FUNCTION_BLOCK FB_Test_Base_Ptr EXTENDS FB_UnitTestBase
VAR_INPUT
END_VAR
VAR_OUTPUT
END_VAR
VAR
END_VAR

(******************************************************************************
Baustein: FB_Test_Base.cleanup
Spezifikation: doc/Spezifikation.pdf, Kap. x.y.z
-------------------------------------------------------------------------------
erstellt:
von:
Geändert:
von:
-------------------------------------------------------------------------------
Beschreibung
Diese Methode...

-------------------------------------------------------------------------------
Input
-

Output
-
******************************************************************************)
METHOD PUBLIC cleanup : BOOL
VAR_INPUT
END_VAR

	cleanup := true;
END_METHOD

(******************************************************************************
Baustein: FB_Test_Base.execute
Spezifikation: doc/Spezifikation.pdf, Kap. x.y.z
-------------------------------------------------------------------------------
erstellt:
von:
Geändert:
von:
-------------------------------------------------------------------------------
Beschreibung
Diese Methode...

-------------------------------------------------------------------------------
Input
-

Output
-
******************************************************************************)
METHOD PUBLIC execute : BOOL
VAR_INPUT
END_VAR
VAR
	bValue1   : ARRAY[0..10] OF BOOL;
	bValue2   : ARRAY[0..10] OF BOOL;
	s8Value1  : ARRAY[0..10] OF SINT;
	s8Value2  : ARRAY[0..10] OF SINT;
	u8Value1  : ARRAY[0..10] OF USINT;
	u8Value2  : ARRAY[0..10] OF USINT;	
	s16Value1 : ARRAY[0..10] OF INT;
	s16Value2 : ARRAY[0..10] OF INT;
	u16Value1 : ARRAY[0..10] OF UINT;
	u16Value2 : ARRAY[0..10] OF UINT;		
	s32Value1 : ARRAY[0..10] OF DINT;
	s32Value2 : ARRAY[0..10] OF DINT;
	u32Value1 : ARRAY[0..10] OF UDINT;
	u32Value2 : ARRAY[0..10] OF UDINT;	
	r32Value1 : ARRAY[0..10] OF REAL;
	r32Value2 : ARRAY[0..10] OF REAL;
	r64Value1 : ARRAY[0..10] OF LREAL;
	r64Value2 : ARRAY[0..10] OF LREAL;
END_VAR


	bValue1[0] := TRUE;
	bValue2[0] := TRUE;
	
	setMessage('Teste Pointer to BOOL equal');
	assertPtrEQUAL(ADR(bValue1[0]), ADR(bValue1[0]));
	
	setMessage('Teste Pointer to BOOL NOT equal');
	assertPtrNOTEQUAL(ADR(bValue1), ADR(bValue2));

(**********************************************) 
	
	s8Value1[0] := 32;
	s8Value2[0] := 32;
	
	setMessage('Teste Pointer to BOOL SINT equal');
	assertPtrEQUAL(ADR(s8Value1[0]), ADR(s8Value1[0]));

	setMessage('Teste Pointer to SINT not equal');
	assertPtrNOTEQUAL(ADR(s8Value1), ADR(s8Value2));
(**********************************************) 	

	u8Value1[0] := 34;
	u8Value2[0] := 34;
	
	setMessage('Teste Pointer to USINT equal');
	assertPtrEQUAL(ADR(u8Value1[0]), ADR(u8Value1[0]));

	setMessage('Teste Pointer to USINT not equal');
	assertPtrNOTEQUAL(ADR(u8Value1), ADR(u8Value2));
(**********************************************) 	
	
	s16Value1[0] := 1323;
	s16Value2[0] := 1323;
	
	setMessage('Teste Pointer to INT equal');
	assertPtrEQUAL(ADR(s16Value1[0]), ADR(s16Value1[0]));

	setMessage('Teste Pointer to INT not equal');
	assertPtrNOTEQUAL(ADR(s16Value1), ADR(s16Value2));
(**********************************************) 	

	u16Value1[0] := 3124;
	u16Value2[0] := 3124;
	
	setMessage('Teste Pointer to UINT equal');
	assertPtrEQUAL(ADR(u16Value1[0]) , ADR(u16Value1[0]) );

	setMessage('Teste Pointer to  UINT not equal');
	assertPtrNOTEQUAL(ADR(u16Value1) , ADR(u16Value2));
(**********************************************) 	

	s32Value1[0] := 1244;
	s32Value2[0] := 1244;
	
	setMessage('Teste Pointer to DINT equal');
	assertPtrEQUAL(ADR(s32Value1[0]), ADR(s32Value1[0]));

	setMessage('Teste Pointer to  DINT not equal');
	assertPtrNOTEQUAL(ADR(s32Value1), ADR(s32Value2));
(**********************************************) 	

	u32Value1[0] := 4344;
	u32Value2[0] := 4344;
	
	setMessage('Teste Pointer to UDINT equal');
	assertPtrEQUAL(ADR(u32Value1[0]), ADR(u32Value1[0]));

	setMessage('Teste Pointer to  UDINT not equal');
	assertPtrNOTEQUAL(ADR(u32Value1), ADR(u32Value2));
(**********************************************) 	

	r32Value1[0] := 133.53245;
	r32Value2[0] := 133.53245;
	
	setMessage('Teste Pointer to REAL equal');
	assertPtrEQUAL(ADR(r32Value1[0]), ADR(r32Value1[0]));

	setMessage('Teste Pointer to  REAL not equal');
	assertPtrNOTEQUAL(ADR(r32Value1), ADR(r32Value2));
(**********************************************) 	

	r64Value1[0] := 1232.53325;
	r64Value2[0] := 1232.53325;

	setMessage('Teste Pointer to LREAL equal');
	assertPtrEQUAL(ADR(r64Value1[0]), ADR(r64Value1[0]));

	setMessage('Teste Pointer to LREAL not equal');
	assertPtrNOTEQUAL(ADR(r64Value1), ADR(r64Value2));

(**********************************************) 	
	execute := TRUE;
END_METHOD

(******************************************************************************
Baustein: FB_Test_Base.prepare
Spezifikation: doc/Spezifikation.pdf, Kap. x.y.z
-------------------------------------------------------------------------------
erstellt:
von:
Geändert:
von:
-------------------------------------------------------------------------------
Beschreibung
Diese Methode...

-------------------------------------------------------------------------------
Input
-

Output
-
******************************************************************************)
METHOD PUBLIC prepare : BOOL
VAR_INPUT
END_VAR

	prepare := true;
END_METHOD

END_FUNCTION_BLOCK

(* stored: Version 1.1.0.1, ProductVersion 3.1.4024.3
   POU FB_Test_Base_Ptr: Id {18af484c-a194-47ec-b09e-eee8a132e9b6}, SpecialFunc None
   Method cleanup: Id {1099d5c5-fa86-441e-94b1-b307d4acd3e2}
   Method execute: Id {8fd83f8a-ddb5-450e-978e-89b220df3e19}
   Method prepare: Id {3232e615-701e-4d31-ba3f-31bec248c2e2} *)
